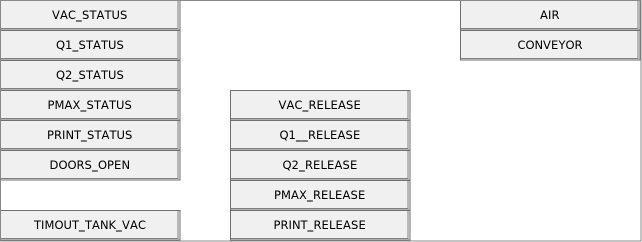
VISUALIZATION FLAGS  // 642x242
    Button (0,0 180x30), "VAC_STATUS", pressed state: Flag_Variables.FLAGS .VAC_STATUS
        toggle Flag_Variables.FLAGS .VAC_STATUS
    Button (0,30 180x30), "Q1_STATUS", pressed state: Flag_Variables.FLAGS .Q1_STATUS
        toggle Flag_Variables.FLAGS .Q1_STATUS
    Button (0,60 180x30), "Q2_STATUS", pressed state: Flag_Variables.FLAGS .Q2_STATUS
        toggle Flag_Variables.FLAGS .Q2_STATUS
    Button (0,90 180x30), "PMAX_STATUS", pressed state: Flag_Variables.FLAGS .PMAX_STATUS
        toggle Flag_Variables.FLAGS .PMAX_STATUS
    Button (0,120 180x30), "PRINT_STATUS", pressed state: Flag_Variables.FLAGS .PRINT_STATUS
        toggle Flag_Variables.FLAGS .PRINT_STATUS
    Button (460,0 180x30), "AIR", pressed state: IOs_Variables.VAC_DO .AIR_VALVE
        toggle IOs_Variables.VAC_DO .AIR_VALVE
    Button (460,30 180x30), "CONVEYOR", pressed state: IOs_Variables.POW_DO .CONVEYOR_RELAIS
        toggle IOs_Variables.POW_DO .CONVEYOR_RELAIS
    Button (230,90 180x30), "VAC_RELEASE", pressed state: Flag_Variables.FLAGS .VAC_RELEASE_CARRIER
        toggle Flag_Variables.FLAGS .VAC_RELEASE_CARRIER
    Button (230,120 180x30), "Q1__RELEASE", pressed state: Flag_Variables.FLAGS .Q1_RELEASE_CARRIER
        toggle Flag_Variables.FLAGS .Q1_RELEASE_CARRIER
    Button (230,150 180x30), "Q2_RELEASE", pressed state: Flag_Variables.FLAGS .Q2_RELEASE_CARRIER
        toggle Flag_Variables.FLAGS .Q2_RELEASE_CARRIER
    Button (230,180 180x30), "PMAX_RELEASE", pressed state: Flag_Variables.FLAGS .PMAX_RELEASE_CARRIER
        toggle Flag_Variables.FLAGS .PMAX_RELEASE_CARRIER
    Button (230,210 180x30), "PRINT_RELEASE", pressed state: Flag_Variables.FLAGS .PRINT_RELEASE_CARRIER
        toggle Flag_Variables.FLAGS .PRINT_RELEASE_CARRIER
    Button (0,150 180x30), "DOORS_OPEN", pressed state: Flag_Variables.FLAGS .DOORS_OPEN
        toggle Flag_Variables.FLAGS .DOORS_OPEN
    Button (0,210 180x30), "TIMOUT_TANK_VAC", pressed state: WATER_TANKS.TIMOUT_TANK_VAC
        toggle WATER_TANKS.TIMOUT_TANK_VAC
END_VISUALIZATION

(* stored: Version 1.1.0.1, ProductVersion 3.1.0.26
   Visu FLAGS: Id {039648ff-bd5c-465e-a4ac-a6f135c70c7f} *)
